// TIA Portal V17 export
// export: Created 2021-12-03T08:13:13.2882669Z, ExportSetting WithDefaults, DisplayName Totally Integrated Automation Portal, DisplayVersion V17, DisplayName TIA Portal Openness, DisplayVersion V17, DisplayName TIA Portal Version Control Interface, DisplayVersion V17, DisplayName STEP 7 Professional, DisplayVersion V17, DisplayName STEP 7 Safety, DisplayVersion V17, DisplayName WinCC Advanced, DisplayVersion V17
FUNCTION_BLOCK "FFB_Simulation"   // FB80, F_FBD
VERSION : 0.1
// stored: AutoNumber false, IsIECCheckEnabled false, UDAEnableTagReadback false
   VAR DB_SPECIFIC
      SimEmSt { ExternalVisible := 'False'; ExternalWritable := 'False'} : Bool;
      SimEnd { ExternalVisible := 'False'; ExternalWritable := 'False'} : Bool;
      Empty : Bool;
   END_VAR
BEGIN

REGION Network 1: Симуляция аварийных кнопок сброс
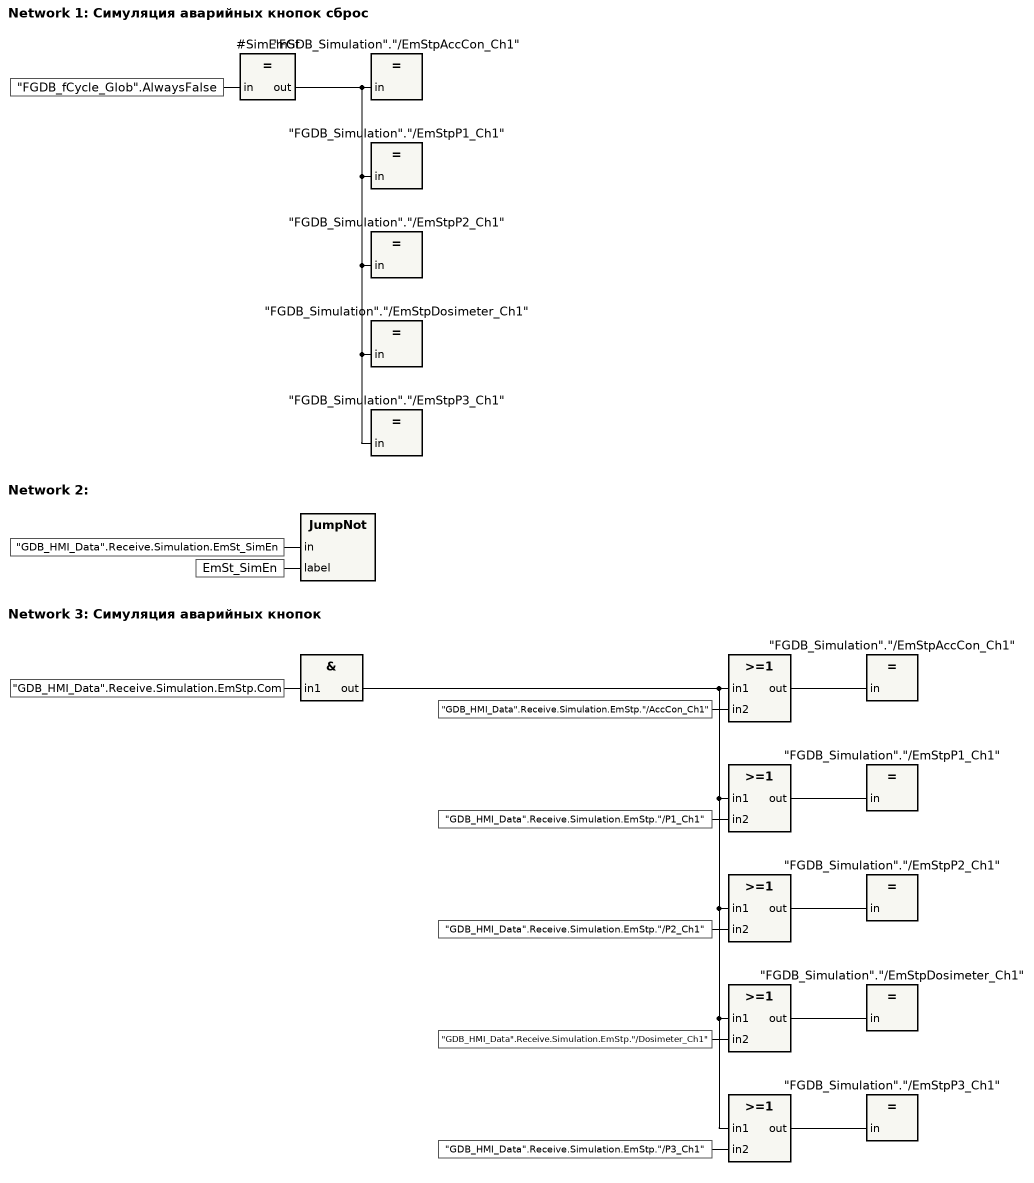
   #SimEmSt := "FGDB_fCycle_Glob".AlwaysFalse;
   "FGDB_Simulation"."/EmStpAccCon_Ch1" := "FGDB_fCycle_Glob".AlwaysFalse;
   "FGDB_Simulation"."/EmStpP1_Ch1" := "FGDB_fCycle_Glob".AlwaysFalse;
   "FGDB_Simulation"."/EmStpP2_Ch1" := "FGDB_fCycle_Glob".AlwaysFalse;
   "FGDB_Simulation"."/EmStpDosimeter_Ch1" := "FGDB_fCycle_Glob".AlwaysFalse;
   "FGDB_Simulation"."/EmStpP3_Ch1" := "FGDB_fCycle_Glob".AlwaysFalse;
END_REGION

REGION Network 2
   // no SCL statement known for JumpNot: written as a call
   JumpNot(in := "GDB_HMI_Data".Receive.Simulation.EmSt_SimEn, label := EmSt_SimEn);
END_REGION

REGION Network 3: Симуляция аварийных кнопок
   "FGDB_Simulation"."/EmStpAccCon_Ch1" := "GDB_HMI_Data".Receive.Simulation.EmStp.Com OR "GDB_HMI_Data".Receive.Simulation.EmStp."/AccCon_Ch1";
   "FGDB_Simulation"."/EmStpP1_Ch1" := "GDB_HMI_Data".Receive.Simulation.EmStp.Com OR "GDB_HMI_Data".Receive.Simulation.EmStp."/P1_Ch1";
   "FGDB_Simulation"."/EmStpP2_Ch1" := "GDB_HMI_Data".Receive.Simulation.EmStp.Com OR "GDB_HMI_Data".Receive.Simulation.EmStp."/P2_Ch1";
   "FGDB_Simulation"."/EmStpDosimeter_Ch1" := "GDB_HMI_Data".Receive.Simulation.EmStp.Com OR "GDB_HMI_Data".Receive.Simulation.EmStp."/Dosimeter_Ch1";
   "FGDB_Simulation"."/EmStpP3_Ch1" := "GDB_HMI_Data".Receive.Simulation.EmStp.Com OR "GDB_HMI_Data".Receive.Simulation.EmStp."/P3_Ch1";
END_REGION

REGION Network 4: Периметр безопасности сброс
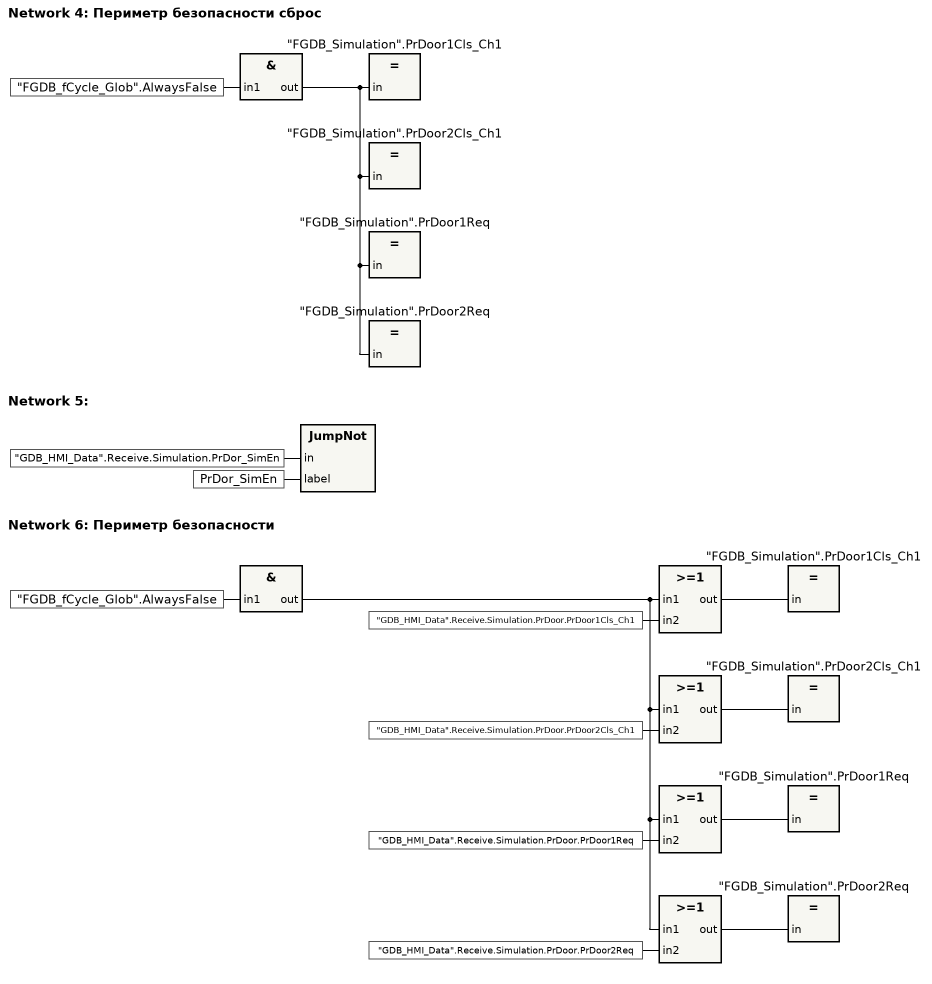
   EmSt_SimEn:
   "FGDB_Simulation".PrDoor1Cls_Ch1 := "FGDB_fCycle_Glob".AlwaysFalse;
   "FGDB_Simulation".PrDoor2Cls_Ch1 := "FGDB_fCycle_Glob".AlwaysFalse;
   "FGDB_Simulation".PrDoor1Req := "FGDB_fCycle_Glob".AlwaysFalse;
   "FGDB_Simulation".PrDoor2Req := "FGDB_fCycle_Glob".AlwaysFalse;
END_REGION

REGION Network 5
   // no SCL statement known for JumpNot: written as a call
   JumpNot(in := "GDB_HMI_Data".Receive.Simulation.PrDor_SimEn, label := PrDor_SimEn);
END_REGION

REGION Network 6: Периметр безопасности
   "FGDB_Simulation".PrDoor1Cls_Ch1 := "FGDB_fCycle_Glob".AlwaysFalse OR "GDB_HMI_Data".Receive.Simulation.PrDoor.PrDoor1Cls_Ch1;
   "FGDB_Simulation".PrDoor2Cls_Ch1 := "FGDB_fCycle_Glob".AlwaysFalse OR "GDB_HMI_Data".Receive.Simulation.PrDoor.PrDoor2Cls_Ch1;
   "FGDB_Simulation".PrDoor1Req := "FGDB_fCycle_Glob".AlwaysFalse OR "GDB_HMI_Data".Receive.Simulation.PrDoor.PrDoor1Req;
   "FGDB_Simulation".PrDoor2Req := "FGDB_fCycle_Glob".AlwaysFalse OR "GDB_HMI_Data".Receive.Simulation.PrDoor.PrDoor2Req;
END_REGION

REGION Network 7: Обратная связь сброс
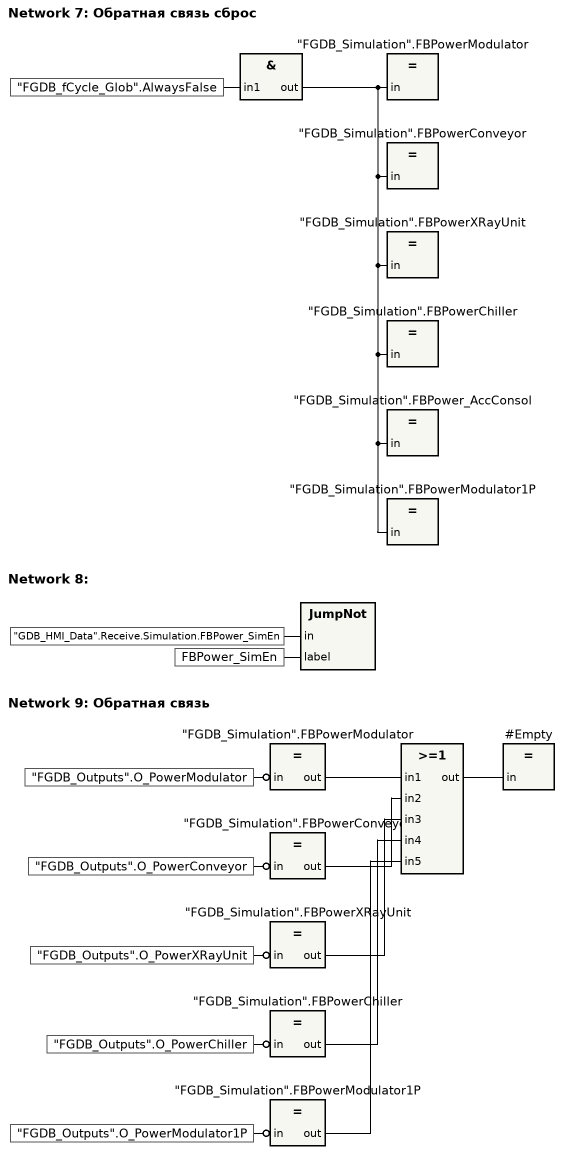
   PrDor_SimEn:
   "FGDB_Simulation".FBPowerModulator := "FGDB_fCycle_Glob".AlwaysFalse;
   "FGDB_Simulation".FBPowerConveyor := "FGDB_fCycle_Glob".AlwaysFalse;
   "FGDB_Simulation".FBPowerXRayUnit := "FGDB_fCycle_Glob".AlwaysFalse;
   "FGDB_Simulation".FBPowerChiller := "FGDB_fCycle_Glob".AlwaysFalse;
   "FGDB_Simulation".FBPower_AccConsol := "FGDB_fCycle_Glob".AlwaysFalse;
   "FGDB_Simulation".FBPowerModulator1P := "FGDB_fCycle_Glob".AlwaysFalse;
END_REGION

REGION Network 8
   // no SCL statement known for JumpNot: written as a call
   JumpNot(in := "GDB_HMI_Data".Receive.Simulation.FBPower_SimEn, label := FBPower_SimEn);
END_REGION

REGION Network 9: Обратная связь
   "FGDB_Simulation".FBPowerModulator := NOT "FGDB_Outputs".O_PowerModulator;
   "FGDB_Simulation".FBPowerConveyor := NOT "FGDB_Outputs".O_PowerConveyor;
   "FGDB_Simulation".FBPowerXRayUnit := NOT "FGDB_Outputs".O_PowerXRayUnit;
   "FGDB_Simulation".FBPowerChiller := NOT "FGDB_Outputs".O_PowerChiller;
   "FGDB_Simulation".FBPowerModulator1P := NOT "FGDB_Outputs".O_PowerModulator1P;
   #Empty := NOT "FGDB_Outputs".O_PowerModulator OR NOT "FGDB_Outputs".O_PowerConveyor OR NOT "FGDB_Outputs".O_PowerXRayUnit OR NOT "FGDB_Outputs".O_PowerChiller OR NOT "FGDB_Outputs".O_PowerModulator1P;
END_REGION

REGION Network 10: симуляция пультов
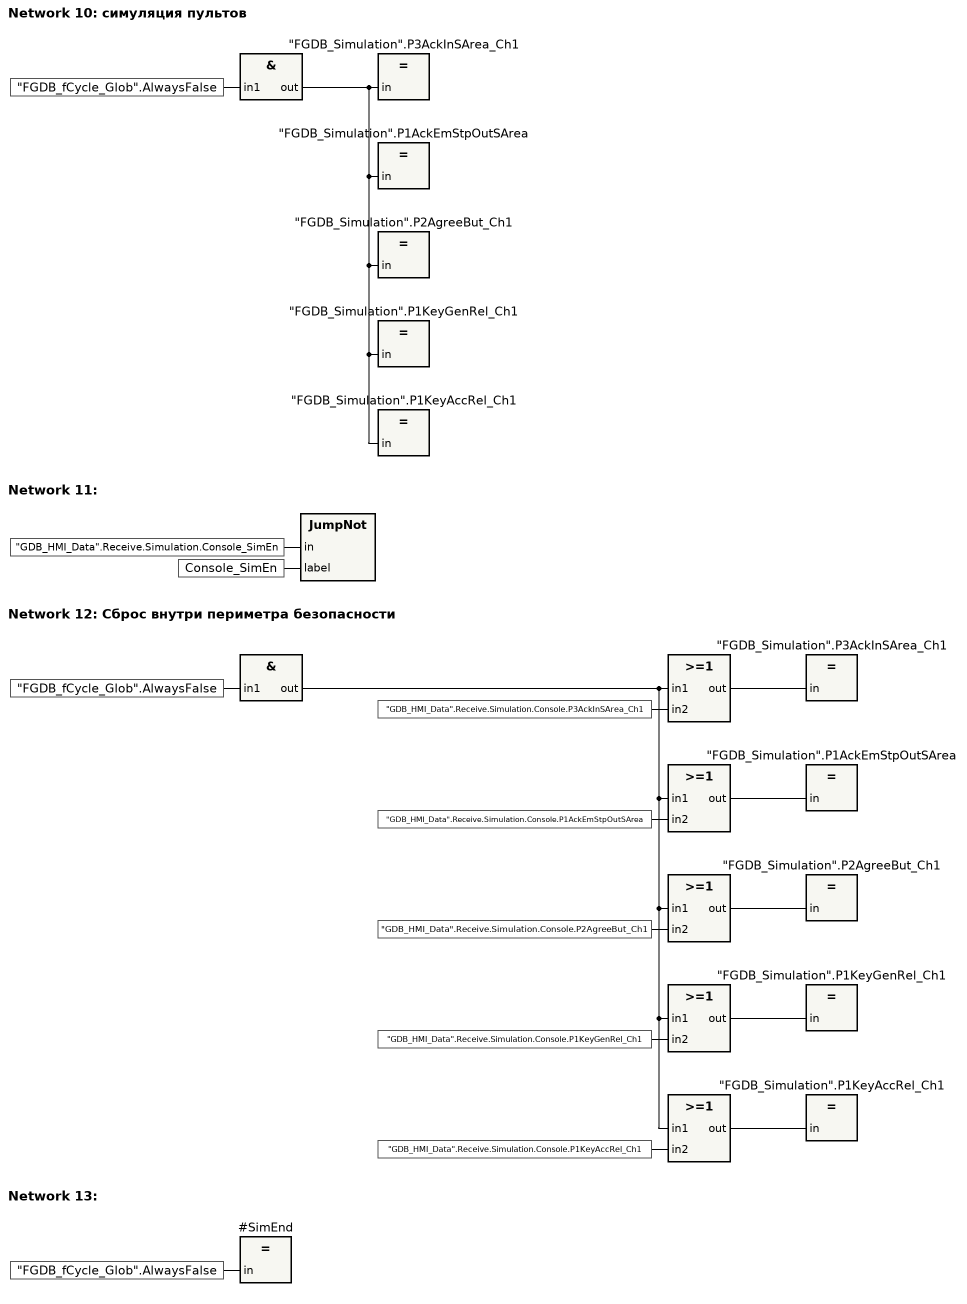
   FBPower_SimEn:
   "FGDB_Simulation".P3AckInSArea_Ch1 := "FGDB_fCycle_Glob".AlwaysFalse;
   "FGDB_Simulation".P1AckEmStpOutSArea := "FGDB_fCycle_Glob".AlwaysFalse;
   "FGDB_Simulation".P2AgreeBut_Ch1 := "FGDB_fCycle_Glob".AlwaysFalse;
   "FGDB_Simulation".P1KeyGenRel_Ch1 := "FGDB_fCycle_Glob".AlwaysFalse;
   "FGDB_Simulation".P1KeyAccRel_Ch1 := "FGDB_fCycle_Glob".AlwaysFalse;
END_REGION

REGION Network 11
   // no SCL statement known for JumpNot: written as a call
   JumpNot(in := "GDB_HMI_Data".Receive.Simulation.Console_SimEn, label := Console_SimEn);
END_REGION

REGION Network 12: Сброс внутри периметра безопасности
   "FGDB_Simulation".P3AckInSArea_Ch1 := "FGDB_fCycle_Glob".AlwaysFalse OR "GDB_HMI_Data".Receive.Simulation.Console.P3AckInSArea_Ch1;
   "FGDB_Simulation".P1AckEmStpOutSArea := "FGDB_fCycle_Glob".AlwaysFalse OR "GDB_HMI_Data".Receive.Simulation.Console.P1AckEmStpOutSArea;
   "FGDB_Simulation".P2AgreeBut_Ch1 := "FGDB_fCycle_Glob".AlwaysFalse OR "GDB_HMI_Data".Receive.Simulation.Console.P2AgreeBut_Ch1;
   "FGDB_Simulation".P1KeyGenRel_Ch1 := "FGDB_fCycle_Glob".AlwaysFalse OR "GDB_HMI_Data".Receive.Simulation.Console.P1KeyGenRel_Ch1;
   "FGDB_Simulation".P1KeyAccRel_Ch1 := "FGDB_fCycle_Glob".AlwaysFalse OR "GDB_HMI_Data".Receive.Simulation.Console.P1KeyAccRel_Ch1;
END_REGION

REGION Network 13
   Console_SimEn:
   #SimEnd := "FGDB_fCycle_Glob".AlwaysFalse;
END_REGION
END_FUNCTION_BLOCK
